Yaskawa INFORM job: TESTWELD.JBI

/JOB
//NAME TESTWELD
///FOLDERNAME IMPORTANT_JOBS
//POS
///NPOS 2,2,0,0,0,0
///TOOL 0
///POSTYPE ROBOT
///RECTAN
///RCONF 0,0,0,0,0,0,0,0,0,0,0,0,0,0,0,0,0,0,0,0,0,0,0,0
C00000=591.981,1055.901,-564.729,53.1276,-25.4002,65.0517
C00001=591.976,1078.761,-564.026,53.1273,-25.4011,65.0523
BC00000=4597.037
BC00001=4597.037
//INST
///DATE 2024/04/16 08:57
///ATTR SC,RW,RJ
////FRAME ROBOT
///GROUP1 RB1,BS1
NOP
MOVL C00000 BC00000 V=11.0
MACRO1 MJ#(0) ARGF24
ARCON
MOVL C00001 BC00001 V=10.0
ARCOF
END
